FUNCTION_BLOCK TwinSAFEGroup IMPLEMENTS ITF_TwinSAFEGroup
VAR
	MySubscribers : ARRAY[0..9] OF ITF_Observer;
	i: INT;
	SubscriberAlreadyAdded : BOOL;
	NumberOfSubscribers: INT;
	ActTwinSAFEState : INT := 8;
	OldTwinSAFEState : INT;
	Update: BOOL;
END_VAR

METHOD Cycle : BOOL
VAR_INPUT
END_VAR
IF ActTwinSAFEState <> OldTwinSAFEState THEN
	OldTwinSAFEState := ActTwinSAFEState;
	This^.Notify();
END_IF
END_METHOD

METHOD GetTwinSAFEState : INT
VAR_INPUT
END_VAR
GetTwinSAFEState := ActTwinSAFEState;
END_METHOD

METHOD PRIVATE Notify : BOOL
VAR_INPUT
END_VAR
FOR i := 0 TO 9 DO
	IF MySubscribers[i] <> 0 THEN
		MySubscribers[i].Update(THIS^);
	END_IF
END_FOR
END_METHOD

METHOD Subscribe : BOOL
VAR_INPUT
	Subscriber : ITF_Observer;
END_VAR
SubscriberAlreadyAdded := FALSE;
FOR i := 0 TO 9 DO
	IF MySubscribers[i] = Subscriber THEN
		SubscriberAlreadyAdded := TRUE;
	END_IF
END_FOR

IF NOT SubscriberAlreadyAdded THEN
	MySubscribers[NumberOfSubscribers] := Subscriber;
	NumberOfSubscribers := NumberOfSubscribers + 1;
END_IF
END_METHOD

METHOD Unsubscribe : BOOL
VAR_INPUT
	Subscriber : ITF_Observer;
END_VAR
FOR i := 0 TO 9 DO
	IF MySubscribers[i] = Subscriber THEN
		MySubscribers[i] := 0;
		NumberOfSubscribers := NumberOfSubscribers - 1;
	END_IF
END_FOR
END_METHOD

END_FUNCTION_BLOCK

(* stored: Version 1.1.0.1, ProductVersion 3.1.4024.12
   POU TwinSAFEGroup: Id {ba0039fd-fd78-4dab-9c52-1edcbf801f38}, SpecialFunc None
   Method Cycle: Id {2e715e96-24c3-407d-a086-b103f22f5a83}
   Method GetTwinSAFEState: Id {0ea0154b-26e0-463d-a391-f024f0b347bb}
   Method Notify: Id {c13b9ce4-d1ad-41a1-99d0-f6df0c7cd297}
   Method Subscribe: Id {1456e187-6826-4e6e-8363-a3082f30d513}
   Method Unsubscribe: Id {797d1020-690c-4b48-98ee-7ff2babc1259} *)
